{attribute addProperty BoxType "ELX9560-0000-0018"}
{attribute addProperty Id "Status_UinAT %I*Status_Uin_51406150810Status_UexAT %I*Status_Uex_A3DD649E810WcStateAT %I*WcState_F855686C1620InfoDataAT %I*InfoData_192954DE1620"}
{attribute addProperty CRC "2208285539"}
{attribute addProperty SizeInBites "48"}
{attribute addProperty SizeInBytes "6"}
TYPE ELX9560_E7D0746E :
STRUCT
	{attribute addProperty Name "Status_Uin"}
	Status_Uin : Status_Uin_51406150;
	{attribute addProperty Name "Status_Uex"}
	Status_Uex : Status_Uex_A3DD649E;
	{attribute addProperty Name "WcState"}
	WcState : WcState_F855686C;
	{attribute addProperty Name "InfoData"}
	InfoData : InfoData_192954DE;
END_STRUCT
END_TYPE

(* stored: Version 1.2.0.0, ProductVersion 3.1.4024.9
   DUT ELX9560_E7D0746E: Id {685c9b11-4beb-46f0-986f-973b3ecfda16} *)
